FUNCTION AGILOG_DEBUG : BOOL
VAR_INPUT
	i_logData : ANY;
	i_printTime :BOOL :=TRUE;
	i_lineBreak :INT :=0;

END_VAR
VAR
	tmpData : LogDataType;
	checkIdx:INT;
END_VAR

IF NOT(GVL_RunTimeLogger.g_enableDebugLog) OR NOT(GVL_RunTimeLogger.g_debugLogReady) THEN
	RETURN;
END_IF

// data decode
tmpData.m_dataType := i_logData.TypeClass;
tmpData.m_dataSize := MIN(i_logData.diSize,96);
tmpData.m_lineBreak := i_lineBreak;
tmpData.m_printTime := i_printTime;
tmpData.m_timeStamp := GVL_RunTimeLogger.g_localSystemTime.systemTime;
MEMCPY(ADR(tmpData.m_data), i_logData.pValue, tmpData.m_dataSize);

FOR checkIdx :=1 TO 20 DO 
	IF TestAndSet(GVL_RunTimeLogger.g_debugLogBufferLock) THEN
		GVL_RunTimeLogger.g_debugLogBuffer[GVL_RunTimeLogger.g_debugLogBufferInPtr] := tmpData;
		// step pointer
		IF GVL_RunTimeLogger.g_debugLogBufferInPtr >= GVL_RunTimeLogger.g_debugLogBufferSize THEN
			GVL_RunTimeLogger.g_debugLogBufferInPtr := 1;
		ELSE
			GVL_RunTimeLogger.g_debugLogBufferInPtr:=GVL_RunTimeLogger.g_debugLogBufferInPtr+1;
		END_IF
		GVL_RunTimeLogger.g_debugLogBufferLock := FALSE;
		EXIT;
	END_IF
END_FOR

END_FUNCTION

(* stored: Version 1.1.0.1, ProductVersion 3.1.4024.11
   POU AGILOG_DEBUG: Id {4d128e6a-b240-42fa-a96e-9a12f0ed4525}, SpecialFunc None *)
